// Mitsubishi GX Works2 project: 프로젝트2-03조   PLC: Q03UDV

// global labels: Global1
VAR_GLOBAL
  공급후진리드 AT X20 : BOOL;
  공급전진리드 AT X21 : BOOL;
  매거진센서 AT X22 : BOOL;
  고주파센서 AT X23 : BOOL;
  용량형센서 AT X24 : BOOL;
  근접포토센서 AT X25 : BOOL;
  그리퍼온리드 AT X27 : BOOL;
  그리퍼오프리드 AT X28 : BOOL;
  물품도착포토 AT X29 : BOOL;
  TG1 AT X2A : BOOL;
  TG2 AT X2B : BOOL;
  TG3 AT X2C : BOOL;
  PB4 AT X2D : BOOL;
  PB5 AT X2E : BOOL;
  창고1 AT X30 : BOOL;
  창고2 AT X31 : BOOL;
  창고3 AT X32 : BOOL;
  창고4 AT X33 : BOOL;
  창고5 AT X34 : BOOL;
  창고6 AT X35 : BOOL;
  창고7 AT X36 : BOOL;
  창고8 AT X37 : BOOL;
  창고9 AT X38 : BOOL;
  도어센서 AT X39 : BOOL;
  압력센서 AT X3A : BOOL;
  공급전솔 AT Y40 : BOOL;
  공급후솔 AT Y41 : BOOL;
  그리퍼온솔 AT Y42 : BOOL;
  그리퍼오프솔 AT Y43 : BOOL;
  경광녹색 AT Y44 : BOOL;
  경광황색 AT Y45 : BOOL;
  경광적색 AT Y46 : BOOL;
  부저 AT Y47 : BOOL;
  컨베이어 AT Y48 : BOOL;
  램프1 AT Y4A : BOOL;
  램프2 AT Y4B : BOOL;
  램프3 AT Y4C : BOOL;
  램프4 AT Y4D : BOOL;
  램프5 AT Y4E : BOOL;
  R그립온명령 AT X1000 : BOOL;
  R그립오프명령 AT X1001 : BOOL;
  R_PLC시작 AT X1002 : BOOL;
  R_판별리셋 AT X1003 : BOOL;
  R재공급 AT X1004 : BOOL;
  R그립온센서 AT Y1000 : BOOL;
  R그립오프센서 AT Y1001 : BOOL;
  R물품없음 AT Y1002 : BOOL;
  R_금속 AT Y1003 : BOOL;
  R_검비금속 AT Y1004 : BOOL;
  R_흰비금속 AT Y1005 : BOOL;
  R물품도착 AT Y1006 : BOOL;
  R컨베이어 AT Y1007 : BOOL;
  R_재시작 AT Y1008 : BOOL;
  R_interrupt AT Y1009 : BOOL;
  R흑전좌 AT Y100A : BOOL;
  R흑전우 AT Y100B : BOOL;
  R흑후좌 AT Y100C : BOOL;
  R흑후우 AT Y100D : BOOL;
  R백전좌 AT Y100E : BOOL;
  R백전우 AT Y100F : BOOL;
  R백후좌 AT Y1010 : BOOL;
  R백후우 AT Y1011 : BOOL;
  R흑전좌완 AT X100A : BOOL;
  R흑전우완 AT X100B : BOOL;
  R흑후좌완 AT X100C : BOOL;
  R흑후우완 AT X100D : BOOL;
  R백전좌완 AT X100E : BOOL;
  R백전우완 AT X100F : BOOL;
  R백후좌완 AT X1010 : BOOL;
  R백후우완 AT X1011 : BOOL;
  R공정종료 AT Y1012 : BOOL;
END_VAR

PROGRAM MAIN
VAR
  t_물품없음 : TIMER;
  시작 : BOOL;
  공급전진 : BOOL;
  공급후진 : BOOL;
  컨베이어온 : BOOL;
  공급종료 : BOOL;
  긴급정지 : BOOL;
  공정종료 : BOOL;
  물품도착 : BOOL;
  재공급 : BOOL;
  C_반복횟수 : COUNTER;
  T_재공급 : TIMER;
  T_물품도착 : TIMER;
  금속 : BOOL;
  흰플라스틱 : BOOL;
  검은플라스틱 : BOOL;
  T_대기 : TIMER;
  검정 : BOOL;
  대기 : BOOL;
  잠시정지 : BOOL;
  T_재기동 : TIMER;
  컨베재기동 : BOOL;
  금속판별 : BOOL;
  물품판별 : BOOL;
  포토센서 : BOOL;
  흰비금속 : BOOL;
  검은비금속 : BOOL;
  t_판별지연 : TIMER;
  컨구동 : BOOL;
  t_컨정지 : TIMER;
  흰색 : BOOL;
  검은색 : BOOL;
END_VAR
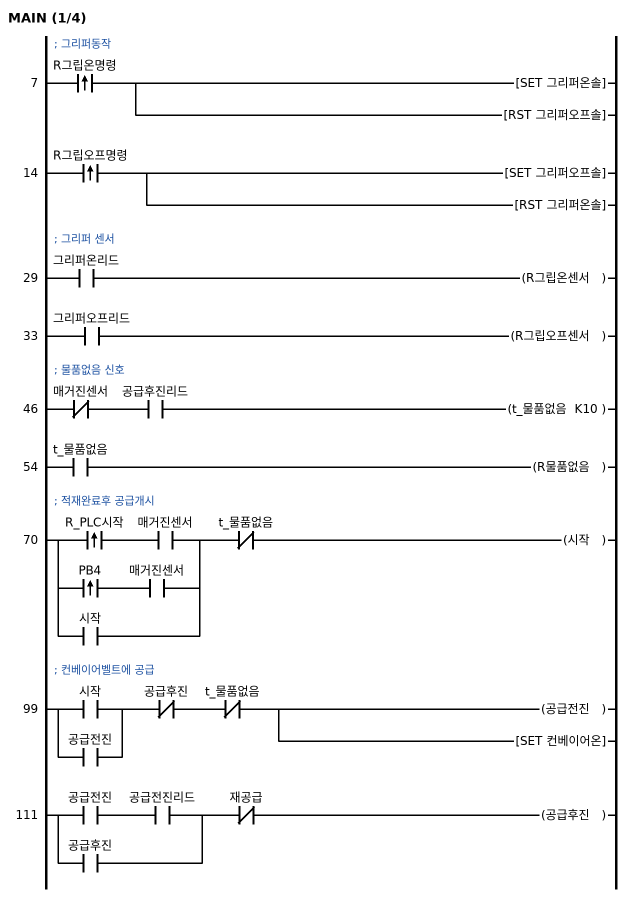
; 그리퍼동작
7     LDP     R그립온명령
      SET     그리퍼온솔
      RST     그리퍼오프솔
14    LDP     R그립오프명령
      SET     그리퍼오프솔
      RST     그리퍼온솔
; 그리퍼 센서
29    LD      그리퍼온리드
      OUT     R그립온센서
33    LD      그리퍼오프리드
      OUT     R그립오프센서
; 물품없음 신호
46    LDI     매거진센서
      AND     공급후진리드
      OUT     t_물품없음 K10
54    LD      t_물품없음
      OUT     R물품없음
; 적재완료후 공급개시
70    LDP     R_PLC시작
      AND     매거진센서
      LDP     PB4
      AND     매거진센서
      ORB
      OR      시작
      ANI     t_물품없음
      OUT     시작
; 컨베이어벨트에 공급
99    LD      시작
      OR      공급전진
      ANI     공급후진
      ANI     t_물품없음
      OUT     공급전진
      SET     컨베이어온
111   LD      공급전진
      AND     공급전진리드
      OR      공급후진
      ANI     재공급
      OUT     공급후진
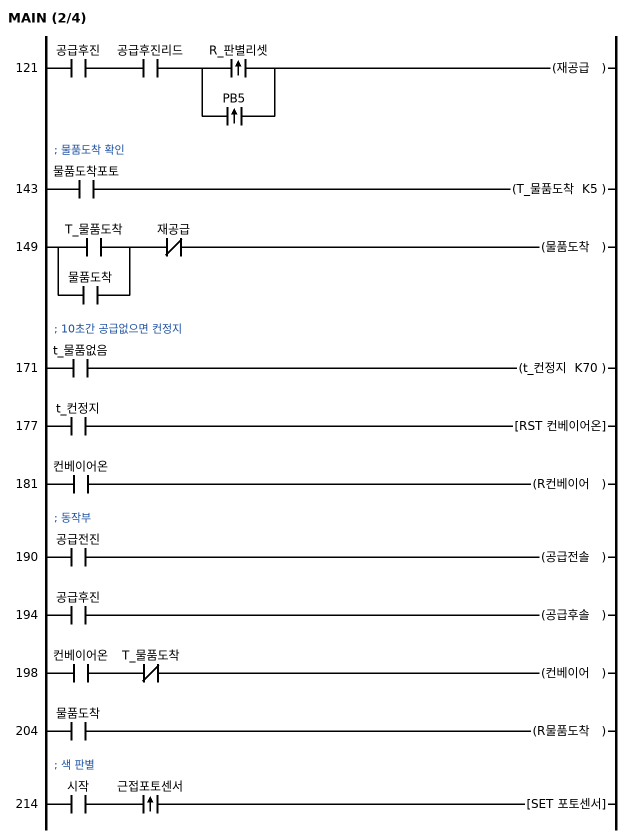
121   LD      공급후진
      AND     공급후진리드
      LDP     R_판별리셋
      ORP     PB5
      ANB
      OUT     재공급
; 물품도착 확인
143   LD      물품도착포토
      OUT     T_물품도착 K5
149   LD      T_물품도착
      OR      물품도착
      ANI     재공급
      OUT     물품도착
; 10초간 공급없으면 컨정지
171   LD      t_물품없음
      OUT     t_컨정지 K70
177   LD      t_컨정지
      RST     컨베이어온
181   LD      컨베이어온
      OUT     R컨베이어
; 동작부
190   LD      공급전진
      OUT     공급전솔
194   LD      공급후진
      OUT     공급후솔
198   LD      컨베이어온
      ANI     T_물품도착
      OUT     컨베이어
204   LD      물품도착
      OUT     R물품도착
; 색 판별
214   LD      시작
      ANDP    근접포토센서
      SET     포토센서
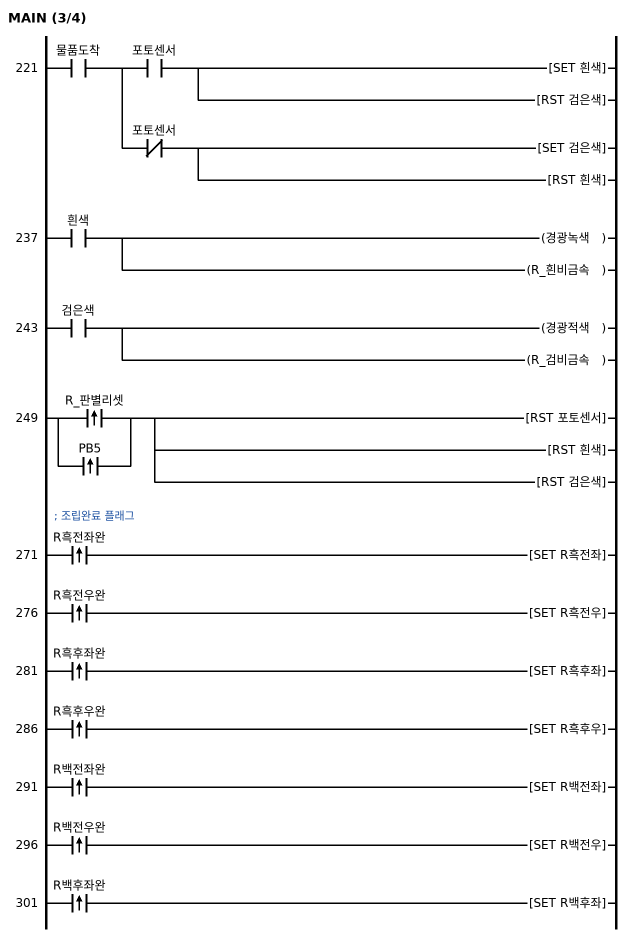
221   LD      물품도착
      MPS
      AND     포토센서
      SET     흰색
      RST     검은색
      MPP
      ANI     포토센서
      SET     검은색
      RST     흰색
237   LD      흰색
      OUT     경광녹색
      OUT     R_흰비금속
243   LD      검은색
      OUT     경광적색
      OUT     R_검비금속
249   LDP     R_판별리셋
      ORP     PB5
      RST     포토센서
      RST     흰색
      RST     검은색
; 조립완료 플래그
271   LDP     R흑전좌완
      SET     R흑전좌
276   LDP     R흑전우완
      SET     R흑전우
281   LDP     R흑후좌완
      SET     R흑후좌
286   LDP     R흑후우완
      SET     R흑후우
291   LDP     R백전좌완
      SET     R백전좌
296   LDP     R백전우완
      SET     R백전우
301   LDP     R백후좌완
      SET     R백후좌
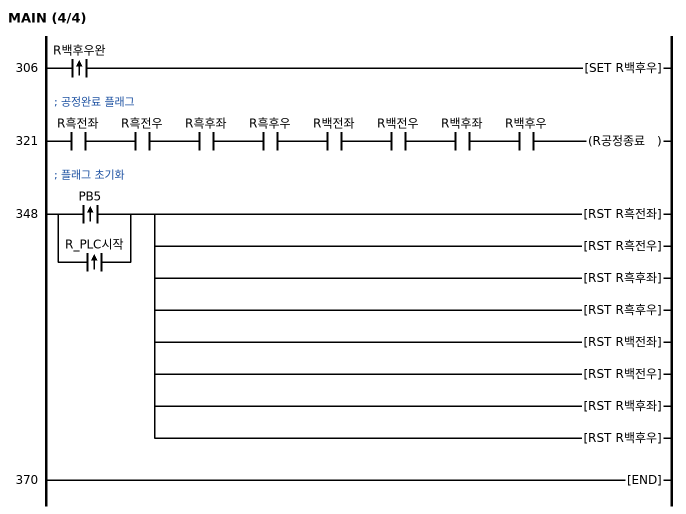
306   LDP     R백후우완
      SET     R백후우
; 공정완료 플래그
321   LD      R흑전좌
      AND     R흑전우
      AND     R흑후좌
      AND     R흑후우
      AND     R백전좌
      AND     R백전우
      AND     R백후좌
      AND     R백후우
      OUT     R공정종료
; 플래그 초기화
348   LDP     PB5
      ORP     R_PLC시작
      RST     R흑전좌
      RST     R흑전우
      RST     R흑후좌
      RST     R흑후우
      RST     R백전좌
      RST     R백전우
      RST     R백후좌
      RST     R백후우
370   END
END_PROGRAM
